// TIA Portal V20 export
TYPE "typeCmHmiInterface"
// stored: Access Published, Namespace Unit1.Em2
   STRUCT
      distance : "LER_typeDistanceInterface";
      softcam : "Unit1.Em2.typeCmHmiInterfaceSoftCam";
      brakeTest : "Unit1.Em2.typeCmHmiInterfaceBrakeTest";
      safeReferencing : "Unit1.Em2.typeCmHmiInterfaceSafeRef";
   END_STRUCT;
   // distance.setValue.direction := TRUE;
   // distance.setValue.distancePTPSV := 6000.0;
END_TYPE
